Universal Robots PolyScope program: grpB222.urp

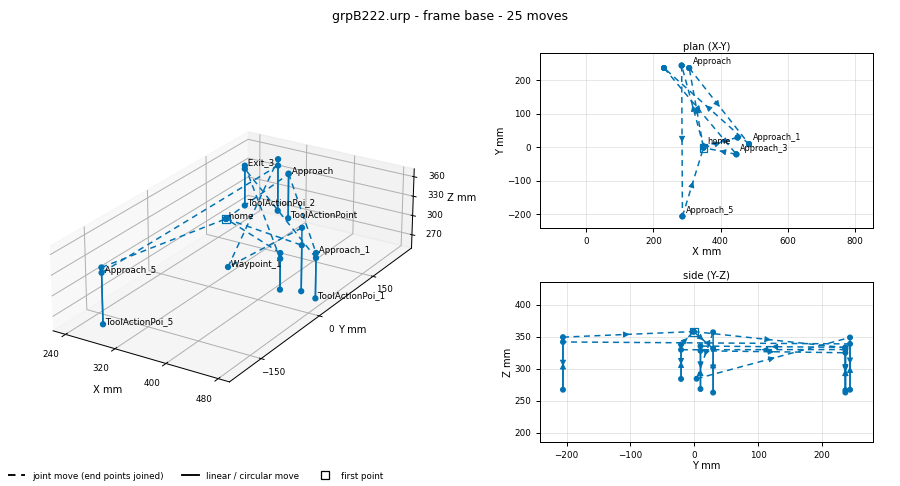
[picture p0: tool path of grpB222.urp in frame base, 25 of 25 moves have a stored position in this frame; points joined in program order, loops and branches not executed]
Program grpB222 (installation=default directory=/programs/Students createdIn=5.11.9.1010452 lastSavedIn=5.11.9.1010452 robotSerialNumber=20225200364)
Calibrated DH parameters: a=[0.00002, -0.569483, -0.54992, -0.00001, -0.000036, 0]; d=[0.180894, -146.691669, 192.918669, -46.053088, 0.119778, 0.115602]; alpha=[1.571425, -0.001534, 0.003359, 1.568739, -1.571477, 0]; deltaTheta=[0, 0.376258, -0.101074, -0.275185, -0.000002, 0]
Robot Program (runOnlyOnce=false)
  MoveJ speed 60 deg/s, acceleration 80 deg/s^2 (useActiveTCP=true) feature=Base
    Waypoint home: TCP in base x=349.211 y=-1.072 z=358.337 mm, rx=2.2343 ry=-2.1885 rz=-0.0245 rad; joints [29.524, -85.445, -128.627, -236.977, -90.829, -151.415] deg
    URCap RG Grip (OnRobot, OnRobot A/S) dataModel(rg-target-force=40.0, rg-target-width=0.1014, Variable(key=on_return, variable(name=on_return)))
    Loop Counting (count=3) loopVariable(name=Loop_1)
      URCap Palletizing (polyscope-pallet-impl, Universal Robots) dataModel(palletFeature=Base, isPalletizing=true, Variable(key=name, variable(name=Pallet_1)), Variable(key=globalCountingVariable, variable(name=Pallet_1_cnt_1, initializeExpression=1)), Variable(key=layerNumberVariable, variable(name=Pallet_1_lno, initializeExpression=1)), Variable(key=layerCountingVariable, variable(name=Pallet_1_lct, initializeExpression=1)), Variable(key=handleSeparatorVariable, variable(name=Pallet_1_sep, initializeExpression=False)), Variable(key=totalCountVariable, variable(name=Pallet_1_tct, initializeExpression=1)), Length(key=objectHeight value=0.00001 unit=M), Variable(key=referencePoint, variable(featureName=referencePoint)), Variable(key=separatorPoint, variable(featureName=separatorPoint))); state(isChildrenLocked=true)
        URCap Patterns (polyscope-pallet-impl, Universal Robots) state(isChildrenLocked=true)
          URCap Pattern (polyscope-pallet-impl, Universal Robots) dataModel(UUID=d454d891-f643-4f11-adf8-96f27634d373, patternType=LINE, objects=3, Variable(key=nameVariable, variable(name=Line_Pattern_1))); state(isChildrenLocked=true)
            URCap Item (polyscope-pallet-impl, Universal Robots) dataModel(UUID=64ea6bed-dd7c-44ae-b121-99742a1ae98b, patternType=LINE, index=0, calibrationDeltaTheta=[-2.1094217540068572E-7, 0.37625772532806073, -0.10107441100396769, -0.2751850025766889, -1.8024952768980196E-6, 2.9402326063437956E-8], calibrationA=[2.0416891277915125E-5, -0.5694828868469309, -0.5499202125525207, -9.504674691390763E-6, -3.603723657207661E-5, 0.0], calibrationD=[0.1808937726775539, -146.69166934821124, 192.91866861971778, -46.05308757405963, 0.11977780403821288, 0.11560212559305974], calibrationAlpha=[1.5714252480212174, -0.0015337665762078037, 0.0033588312559612306, 1.5687392298942362, -1.5714772428732047, 0.0], calibrationJointChecksum=[-1490546360, -1456574554, -1506622700, -1493399207, -1492840923, -1492940558], calibrationStatus=2, calibrationValidChecksum=true, baseToFeature=[0.0, 0.0, 0.0, 0.0, 0.0, 0.0], TCPOffset=[-6.479107609730361E-6, -2.1640648664167372E-6, 6.459965172400661E-6, -7.466567837094426E-7, 6.496160494327226E-6, 1.4031189272003694E-5], Variable(key=variable, variable(name=StartItem_1)), JointPositions(key=jointpositions, JointPosition(key=[1], Angle(key=pos value=1.117784 unit=RAD)), JointPosition(key=[2], Angle(key=pos value=-1.682038 unit=RAD)), JointPosition(key=[3], Angle(key=pos value=-2.256967 unit=RAD)), JointPosition(key=[4], Angle(key=pos value=-3.923758 unit=RAD)), JointPosition(key=[5], Angle(key=pos value=-1.592734 unit=RAD)), JointPosition(key=[6], Angle(key=pos value=-2.039439 unit=RAD))))
            URCap Item (polyscope-pallet-impl, Universal Robots) dataModel(UUID=acc9778f-9bc3-49a4-a915-6e2dc52f2b95, patternType=LINE, index=1, calibrationDeltaTheta=[-2.1094217540068572E-7, 0.37625772532806073, -0.10107441100396769, -0.2751850025766889, -1.8024952768980196E-6, 2.9402326063437956E-8], calibrationA=[2.0416891277915125E-5, -0.5694828868469309, -0.5499202125525207, -9.504674691390763E-6, -3.603723657207661E-5, 0.0], calibrationD=[0.1808937726775539, -146.69166934821124, 192.91866861971778, -46.05308757405963, 0.11977780403821288, 0.11560212559305974], calibrationAlpha=[1.5714252480212174, -0.0015337665762078037, 0.0033588312559612306, 1.5687392298942362, -1.5714772428732047, 0.0], calibrationJointChecksum=[-1490546360, -1456574554, -1506622700, -1493399207, -1492840923, -1492940558], calibrationStatus=2, calibrationValidChecksum=true, baseToFeature=[0.0, 0.0, 0.0, 0.0, 0.0, 0.0], TCPOffset=[1.9374486620010734E-5, 1.7322688802723363E-5, 1.403770617985911E-5, -2.993389842851144E-5, 5.83636955800167E-5, -2.7174622035027854E-5], Variable(key=variable, variable(name=EndItem_1)), JointPositions(key=jointpositions, JointPosition(key=[1], Angle(key=pos value=1.274188 unit=RAD)), JointPosition(key=[2], Angle(key=pos value=-1.609872 unit=RAD)), JointPosition(key=[3], Angle(key=pos value=-2.336948 unit=RAD)), JointPosition(key=[4], Angle(key=pos value=-3.912921 unit=RAD)), JointPosition(key=[5], Angle(key=pos value=-1.593886 unit=RAD)), JointPosition(key=[6], Angle(key=pos value=-1.883026 unit=RAD))))
        URCap Layers (polyscope-pallet-impl, Universal Robots) dataModel(separators=[false], selectedPatterns=[d454d891-f643-4f11-adf8-96f27634d373])
        URCap At Each Item (polyscope-pallet-impl, Universal Robots) dataModel(selectedPattern=d454d891-f643-4f11-adf8-96f27634d373, selectedPosition=64ea6bed-dd7c-44ae-b121-99742a1ae98b, Approach_calibrationDeltaTheta=[-2.1094217540068572E-7, 0.37625772532806073, -0.10107441100396769, -0.2751850025766889, -1.8024952768980196E-6, 2.9402326063437956E-8], Approach_calibrationA=[2.0416891277915125E-5, -0.5694828868469309, -0.5499202125525207, -9.504674691390763E-6, -3.603723657207661E-5, 0.0], Approach_calibrationD=[0.1808937726775539, -146.69166934821124, 192.91866861971778, -46.05308757405963, 0.11977780403821288, 0.11560212559305974], Approach_calibrationAlpha=[1.5714252480212174, -0.0015337665762078037, 0.0033588312559612306, 1.5687392298942362, -1.5714772428732047, 0.0], Approach_calibrationJointChecksum=[-1490546360, -1456574554, -1506622700, -1493399207, -1492840923, -1492940558], Approach_calibrationStatus=2, Approach_calibrationValidChecksum=true, Approach_baseToFeature=[0.0, 0.0, 0.0, 0.0, 0.0, 0.0], Approach_TCPOffset=[2.5781352005288527E-5, 2.5671739316002196E-6, 1.3650458078329208E-5, -3.390166594725408E-5, 6.308214025204194E-5, 7.147033976335445E-5], Exit_calibrationDeltaTheta=[-2.1094217540068572E-7, 0.37625772532806073, -0.10107441100396769, -0.2751850025766889, -1.8024952768980196E-6, 2.9402326063437956E-8], Exit_calibrationA=[2.0416891277915125E-5, -0.5694828868469309, -0.5499202125525207, -9.504674691390763E-6, -3.603723657207661E-5, 0.0], Exit_calibrationD=[0.1808937726775539, -146.69166934821124, 192.91866861971778, -46.05308757405963, 0.11977780403821288, 0.11560212559305974], Exit_calibrationAlpha=[1.5714252480212174, -0.0015337665762078037, 0.0033588312559612306, 1.5687392298942362, -1.5714772428732047, 0.0], Exit_calibrationJointChecksum=[-1490546360, -1456574554, -1506622700, -1493399207, -1492840923, -1492940558], Exit_calibrationStatus=2, Exit_calibrationValidChecksum=true, Exit_baseToFeature=[0.0, 0.0, 0.0, 0.0, 0.0, 0.0], Exit_TCPOffset=[4.769778841942629E-5, 1.539205112810471E-5, 1.24869559859353E-5, -7.939274321106401E-5, 8.864952215778513E-5, 6.565241233819079E-5], currentWizardState=SHOW_DONE, Pose(key=refBaseToFeature, Position(key=posePosition, Length(key=X value=0 unit=M), Length(key=Y value=0 unit=M), Length(key=Z value=0 unit=M)), Rotation(key=poseRotation, Angle(key=RX value=0 unit=RAD), Angle(key=RY value=0 unit=RAD), Angle(key=RZ value=0 unit=RAD))), Pose(key=refPose, Position(key=posePosition, Length(key=X value=0.306641 unit=M), Length(key=Y value=0.236656 unit=M), Length(key=Z value=0.26283 unit=M)), Rotation(key=poseRotation, Angle(key=RX value=2.234367 unit=RAD), Angle(key=RY value=-2.188526 unit=RAD), Angle(key=RZ value=-0.024467 unit=RAD))), JointPositions(key=Approach_jointpositions, JointPosition(key=[1], Angle(key=pos value=1.117614 unit=RAD)), JointPosition(key=[2], Angle(key=pos value=-1.591367 unit=RAD)), JointPosition(key=[3], Angle(key=pos value=-2.200898 unit=RAD)), JointPosition(key=[4], Angle(key=pos value=-4.07051 unit=RAD)), JointPosition(key=[5], Angle(key=pos value=-1.593074 unit=RAD)), JointPosition(key=[6], Angle(key=pos value=-2.040098 unit=RAD))), JointPositions(key=Exit_jointpositions, JointPosition(key=[1], Angle(key=pos value=1.117612 unit=RAD)), JointPosition(key=[2], Angle(key=pos value=-1.590509 unit=RAD)), JointPosition(key=[3], Angle(key=pos value=-2.200233 unit=RAD)), JointPosition(key=[4], Angle(key=pos value=-4.072033 unit=RAD)), JointPosition(key=[5], Angle(key=pos value=-1.593077 unit=RAD)), JointPosition(key=[6], Angle(key=pos value=-2.040105 unit=RAD))))
          URCap Generated Movements (polyscope-pallet-impl, Universal Robots) state(isChildrenLocked=true)
            MoveJ speed 60 deg/s, acceleration 80 deg/s^2 (useActiveTCP=true) feature=referencePoint
              Waypoint Approach: TCP in base x=306.638 y=236.63 z=332.959 mm, rx=2.2342 ry=-2.1886 rz=-0.0244 rad; joints [64.033, -91.179, -126.104, -233.224, -91.277, -116.887] deg; TCP offset x=0 y=0 z=0 mm, rx=0 ry=0 rz=0 rad; feature pose in base x=306.641 y=236.656 z=262.83 mm, rx=2.2344 ry=-2.1885 rz=-0.0245 rad
            MoveL speed 250 mm/s, acceleration 1200 mm/s^2 (useActiveTCP=true) feature(featureName=referencePoint)
              Waypoint ToolActionPoint: TCP in base x=306.641 y=236.656 z=262.83 mm, rx=2.2344 ry=-2.1885 rz=-0.0245 rad; joints [64.045, -96.692, -129.469, -224.342, -91.256, -116.849] deg; TCP offset x=0 y=0 z=0 mm, rx=0 ry=0 rz=0 rad
            Folder Tool action
              URCap RG Grip (OnRobot, OnRobot A/S) dataModel(rg-target-force=40.0, rg-target-width=0.0747)
            MoveL speed 250 mm/s, acceleration 1200 mm/s^2 (useActiveTCP=true) feature(featureName=referencePoint)
              Waypoint Exit_1: TCP in base x=306.626 y=236.608 z=333.664 mm, rx=2.2342 ry=-2.1885 rz=-0.0245 rad; joints [64.033, -91.128, -126.068, -233.314, -91.278, -116.888] deg; TCP offset x=0 y=0 z=0 mm, rx=0 ry=0 rz=0 rad
      URCap Palletizing (polyscope-pallet-impl, Universal Robots) dataModel(palletFeature=Base, isPalletizing=true, Length(key=objectHeight value=0.00001 unit=M), Variable(key=name, variable(name=Pallet_2)), Variable(key=globalCountingVariable, variable(name=Pallet_2_cnt, initializeExpression=1)), Variable(key=layerNumberVariable, variable(name=Pallet_2_lno, initializeExpression=1)), Variable(key=layerCountingVariable, variable(name=Pallet_2_lct, initializeExpression=1)), Variable(key=handleSeparatorVariable, variable(name=Pallet_2_sep, initializeExpression=False)), Variable(key=totalCountVariable, variable(name=Pallet_2_tct, initializeExpression=1)), Variable(key=referencePoint, variable(featureName=referencePoin_1)), Variable(key=separatorPoint, variable(featureName=separatorPoin_1))); state(isChildrenLocked=true)
        URCap Patterns (polyscope-pallet-impl, Universal Robots) state(isChildrenLocked=true)
          URCap Pattern (polyscope-pallet-impl, Universal Robots) dataModel(UUID=45a8ee5b-4a8a-4b28-a838-296028420bac, patternType=LINE, objects=3, Variable(key=nameVariable, variable(name=Line_Pattern_2))); state(isChildrenLocked=true)
            URCap Item (polyscope-pallet-impl, Universal Robots) dataModel(UUID=b27af457-f974-4cfa-a6aa-9b6048d656b7, patternType=LINE, index=0, calibrationDeltaTheta=[-2.1094217540068572E-7, 0.37625772532806073, -0.10107441100396769, -0.2751850025766889, -1.8024952768980196E-6, 2.9402326063437956E-8], calibrationA=[2.0416891277915125E-5, -0.5694828868469309, -0.5499202125525207, -9.504674691390763E-6, -3.603723657207661E-5, 0.0], calibrationD=[0.1808937726775539, -146.69166934821124, 192.91866861971778, -46.05308757405963, 0.11977780403821288, 0.11560212559305974], calibrationAlpha=[1.5714252480212174, -0.0015337665762078037, 0.0033588312559612306, 1.5687392298942362, -1.5714772428732047, 0.0], calibrationJointChecksum=[-1490546360, -1456574554, -1506622700, -1493399207, -1492840923, -1492940558], calibrationStatus=2, calibrationValidChecksum=true, baseToFeature=[0.0, 0.0, 0.0, 0.0, 0.0, 0.0], TCPOffset=[6.044463015194733E-8, 8.449471585958435E-6, 1.7500404647985413E-5, -5.2372560383104365E-6, 3.613439746095069E-5, 5.677349546775118E-6], Variable(key=variable, variable(name=StartItem_2)), JointPositions(key=jointpositions, JointPosition(key=[1], Angle(key=pos value=0.387931 unit=RAD)), JointPosition(key=[2], Angle(key=pos value=-1.834321 unit=RAD)), JointPosition(key=[3], Angle(key=pos value=-2.075058 unit=RAD)), JointPosition(key=[4], Angle(key=pos value=-3.964125 unit=RAD)), JointPosition(key=[5], Angle(key=pos value=-1.582177 unit=RAD)), JointPosition(key=[6], Angle(key=pos value=-2.769248 unit=RAD))))
            URCap Item (polyscope-pallet-impl, Universal Robots) dataModel(UUID=9365cefe-048c-485e-b644-eb1a72d9b5fb, patternType=LINE, index=1, calibrationDeltaTheta=[-2.1094217540068572E-7, 0.37625772532806073, -0.10107441100396769, -0.2751850025766889, -1.8024952768980196E-6, 2.9402326063437956E-8], calibrationA=[2.0416891277915125E-5, -0.5694828868469309, -0.5499202125525207, -9.504674691390763E-6, -3.603723657207661E-5, 0.0], calibrationD=[0.1808937726775539, -146.69166934821124, 192.91866861971778, -46.05308757405963, 0.11977780403821288, 0.11560212559305974], calibrationAlpha=[1.5714252480212174, -0.0015337665762078037, 0.0033588312559612306, 1.5687392298942362, -1.5714772428732047, 0.0], calibrationJointChecksum=[-1490546360, -1456574554, -1506622700, -1493399207, -1492840923, -1492940558], calibrationStatus=2, calibrationValidChecksum=true, baseToFeature=[0.0, 0.0, 0.0, 0.0, 0.0, 0.0], TCPOffset=[-2.5050077170275797E-5, -1.1405127266772563E-5, 6.504272814233936E-7, 1.2865247891813043E-5, -3.7242278860020355E-5, -5.7602559931804165E-5], JointPositions(key=jointpositions, JointPosition(key=[1], Angle(key=pos value=0.44248 unit=RAD)), JointPosition(key=[2], Angle(key=pos value=-1.741933 unit=RAD)), JointPosition(key=[3], Angle(key=pos value=-2.182688 unit=RAD)), JointPosition(key=[4], Angle(key=pos value=-3.948526 unit=RAD)), JointPosition(key=[5], Angle(key=pos value=-1.583418 unit=RAD)), JointPosition(key=[6], Angle(key=pos value=-2.714732 unit=RAD))), Variable(key=variable, variable(name=EndItem_2)))
        URCap Layers (polyscope-pallet-impl, Universal Robots) dataModel(separators=[false], selectedPatterns=[45a8ee5b-4a8a-4b28-a838-296028420bac])
        URCap At Each Item (polyscope-pallet-impl, Universal Robots) dataModel(selectedPattern=45a8ee5b-4a8a-4b28-a838-296028420bac, selectedPosition=b27af457-f974-4cfa-a6aa-9b6048d656b7, Approach_calibrationDeltaTheta=[-2.1094217540068572E-7, 0.37625772532806073, -0.10107441100396769, -0.2751850025766889, -1.8024952768980196E-6, 2.9402326063437956E-8], Approach_calibrationA=[2.0416891277915125E-5, -0.5694828868469309, -0.5499202125525207, -9.504674691390763E-6, -3.603723657207661E-5, 0.0], Approach_calibrationD=[0.1808937726775539, -146.69166934821124, 192.91866861971778, -46.05308757405963, 0.11977780403821288, 0.11560212559305974], Approach_calibrationAlpha=[1.5714252480212174, -0.0015337665762078037, 0.0033588312559612306, 1.5687392298942362, -1.5714772428732047, 0.0], Approach_calibrationJointChecksum=[-1490546360, -1456574554, -1506622700, -1493399207, -1492840923, -1492940558], Approach_calibrationStatus=2, Approach_calibrationValidChecksum=true, Approach_baseToFeature=[0.0, 0.0, 0.0, 0.0, 0.0, 0.0], Approach_TCPOffset=[2.1697404932576178E-5, 2.6992522534685648E-5, 2.5750409892999482E-5, -7.803021143395113E-5, 1.3046438018846386E-5, 5.729013140880056E-5], Exit_calibrationDeltaTheta=[-2.1094217540068572E-7, 0.37625772532806073, -0.10107441100396769, -0.2751850025766889, -1.8024952768980196E-6, 2.9402326063437956E-8], Exit_calibrationA=[2.0416891277915125E-5, -0.5694828868469309, -0.5499202125525207, -9.504674691390763E-6, -3.603723657207661E-5, 0.0], Exit_calibrationD=[0.1808937726775539, -146.69166934821124, 192.91866861971778, -46.05308757405963, 0.11977780403821288, 0.11560212559305974], Exit_calibrationAlpha=[1.5714252480212174, -0.0015337665762078037, 0.0033588312559612306, 1.5687392298942362, -1.5714772428732047, 0.0], Exit_calibrationJointChecksum=[-1490546360, -1456574554, -1506622700, -1493399207, -1492840923, -1492940558], Exit_calibrationStatus=2, Exit_calibrationValidChecksum=true, Exit_baseToFeature=[0.0, 0.0, 0.0, 0.0, 0.0, 0.0], Exit_TCPOffset=[1.9248975832635864E-5, 2.1285860685449354E-5, 4.198514513409357E-5, -9.050769865031771E-5, 5.440701917327053E-5, 1.0746634104783018E-6], currentWizardState=LANDING, Pose(key=refBaseToFeature, Position(key=posePosition, Length(key=X value=0 unit=M), Length(key=Y value=0 unit=M), Length(key=Z value=0 unit=M)), Rotation(key=poseRotation, Angle(key=RX value=0 unit=RAD), Angle(key=RY value=0 unit=RAD), Angle(key=RZ value=0 unit=RAD))), Pose(key=refPose, Position(key=posePosition, Length(key=X value=0.484958 unit=M), Length(key=Y value=0.009632 unit=M), Length(key=Z value=0.268373 unit=M)), Rotation(key=poseRotation, Angle(key=RX value=2.234217 unit=RAD), Angle(key=RY value=-2.1886 unit=RAD), Angle(key=RZ value=-0.024602 unit=RAD))), JointPositions(key=Approach_jointpositions, JointPosition(key=[1], Angle(key=pos value=0.384856 unit=RAD)), JointPosition(key=[2], Angle(key=pos value=-1.753755 unit=RAD)), JointPosition(key=[3], Angle(key=pos value=-2.013529 unit=RAD)), JointPosition(key=[4], Angle(key=pos value=-4.106379 unit=RAD)), JointPosition(key=[5], Angle(key=pos value=-1.582524 unit=RAD)), JointPosition(key=[6], Angle(key=pos value=-2.772795 unit=RAD))), JointPositions(key=Exit_jointpositions, JointPosition(key=[1], Angle(key=pos value=0.384867 unit=RAD)), JointPosition(key=[2], Angle(key=pos value=-1.761546 unit=RAD)), JointPosition(key=[3], Angle(key=pos value=-2.019642 unit=RAD)), JointPosition(key=[4], Angle(key=pos value=-4.092474 unit=RAD)), JointPosition(key=[5], Angle(key=pos value=-1.582497 unit=RAD)), JointPosition(key=[6], Angle(key=pos value=-2.772737 unit=RAD))))
          URCap Generated Movements (polyscope-pallet-impl, Universal Robots) state(isChildrenLocked=true)
            MoveJ speed 60 deg/s, acceleration 80 deg/s^2 (useActiveTCP=true) feature=referencePoin_1
              Waypoint Approach_1: TCP in base x=484.931 y=9.61 z=335.59 mm, rx=2.2341 ry=-2.1886 rz=-0.0247 rad; joints [22.049, -100.483, -115.371, -235.278, -90.673, -158.868] deg; TCP offset x=0 y=0 z=0 mm, rx=0 ry=0 rz=0 rad; feature pose in base x=484.958 y=9.632 z=268.373 mm, rx=2.2342 ry=-2.1886 rz=-0.0246 rad
            MoveL speed 250 mm/s, acceleration 1200 mm/s^2 (useActiveTCP=true) feature(featureName=referencePoin_1)
              Waypoint ToolActionPoi_1: TCP in base x=484.958 y=9.632 z=268.373 mm, rx=2.2342 ry=-2.1886 rz=-0.0246 rad; joints [22.056, -104.961, -118.259, -227.907, -90.656, -158.84] deg; TCP offset x=0 y=0 z=0 mm, rx=0 ry=0 rz=0 rad
            Folder Tool action
              URCap RG Grip (OnRobot, OnRobot A/S) dataModel(rg-target-force=40.0, rg-target-width=0.1014)
            MoveL speed 250 mm/s, acceleration 1200 mm/s^2 (useActiveTCP=true) feature(featureName=referencePoin_1)
              Waypoint Exit_2: TCP in base x=484.936 y=9.612 z=328.275 mm, rx=2.2341 ry=-2.1885 rz=-0.0246 rad; joints [22.05, -100.931, -115.721, -234.481, -90.669, -158.867] deg; TCP offset x=0 y=0 z=0 mm, rx=0 ry=0 rz=0 rad
    Loop Counting (count=3) loopVariable(name=Loop_2)
      URCap Palletizing (polyscope-pallet-impl, Universal Robots) dataModel(palletFeature=Base, isPalletizing=true, Length(key=objectHeight value=0.00001 unit=M), Variable(key=name, variable(name=Pallet_3)), Variable(key=globalCountingVariable, variable(name=Pallet_3_cnt, initializeExpression=1)), Variable(key=layerNumberVariable, variable(name=Pallet_3_lno, initializeExpression=1)), Variable(key=layerCountingVariable, variable(name=Pallet_3_lct, initializeExpression=1)), Variable(key=handleSeparatorVariable, variable(name=Pallet_3_sep, initializeExpression=False)), Variable(key=totalCountVariable, variable(name=Pallet_3_tct, initializeExpression=1)), Variable(key=referencePoint, variable(featureName=referencePoin_2)), Variable(key=separatorPoint, variable(featureName=separatorPoin_2))); state(isChildrenLocked=true)
        URCap Patterns (polyscope-pallet-impl, Universal Robots) state(isChildrenLocked=true)
          URCap Pattern (polyscope-pallet-impl, Universal Robots) dataModel(UUID=2b4160e0-b2a1-4967-a814-10dbe05e682f, patternType=LINE, objects=3, Variable(key=nameVariable, variable(name=Line_Pattern_3))); state(isChildrenLocked=true)
            URCap Item (polyscope-pallet-impl, Universal Robots) dataModel(UUID=27d7fe94-2af4-48ef-bc96-4bf19b8c453b, patternType=LINE, index=0, calibrationDeltaTheta=[-2.1094217540068572E-7, 0.37625772532806073, -0.10107441100396769, -0.2751850025766889, -1.8024952768980196E-6, 2.9402326063437956E-8], calibrationA=[2.0416891277915125E-5, -0.5694828868469309, -0.5499202125525207, -9.504674691390763E-6, -3.603723657207661E-5, 0.0], calibrationD=[0.1808937726775539, -146.69166934821124, 192.91866861971778, -46.05308757405963, 0.11977780403821288, 0.11560212559305974], calibrationAlpha=[1.5714252480212174, -0.0015337665762078037, 0.0033588312559612306, 1.5687392298942362, -1.5714772428732047, 0.0], calibrationJointChecksum=[-1490546360, -1456574554, -1506622700, -1493399207, -1492840923, -1492940558], calibrationStatus=2, calibrationValidChecksum=true, baseToFeature=[0.0, 0.0, 0.0, 0.0, 0.0, 0.0], TCPOffset=[-1.591908718442947E-5, -1.0217043891230793E-5, -2.3879269327009567E-5, 3.6458983264753285E-5, -3.8288802833761E-5, -2.268284047652254E-6], JointPositions(key=jointpositions, JointPosition(key=[1], Angle(key=pos value=1.343103 unit=RAD)), JointPosition(key=[2], Angle(key=pos value=-1.581886 unit=RAD)), JointPosition(key=[3], Angle(key=pos value=-2.365664 unit=RAD)), JointPosition(key=[4], Angle(key=pos value=-3.910843 unit=RAD)), JointPosition(key=[5], Angle(key=pos value=-1.594245 unit=RAD)), JointPosition(key=[6], Angle(key=pos value=-1.814135 unit=RAD))), Variable(key=variable, variable(name=StartItem_3)))
            URCap Item (polyscope-pallet-impl, Universal Robots) dataModel(UUID=072fc38f-4205-41de-a57f-9e135fb71f30, patternType=LINE, index=1, calibrationDeltaTheta=[-2.1094217540068572E-7, 0.37625772532806073, -0.10107441100396769, -0.2751850025766889, -1.8024952768980196E-6, 2.9402326063437956E-8], calibrationA=[2.0416891277915125E-5, -0.5694828868469309, -0.5499202125525207, -9.504674691390763E-6, -3.603723657207661E-5, 0.0], calibrationD=[0.1808937726775539, -146.69166934821124, 192.91866861971778, -46.05308757405963, 0.11977780403821288, 0.11560212559305974], calibrationAlpha=[1.5714252480212174, -0.0015337665762078037, 0.0033588312559612306, 1.5687392298942362, -1.5714772428732047, 0.0], calibrationJointChecksum=[-1490546360, -1456574554, -1506622700, -1493399207, -1492840923, -1492940558], calibrationStatus=2, calibrationValidChecksum=true, baseToFeature=[0.0, 0.0, 0.0, 0.0, 0.0, 0.0], TCPOffset=[-9.716888572375293E-7, -8.226545365752624E-6, -1.2344780305817427E-5, 2.4931859189616642E-5, -3.857283165511878E-5, 3.9017410809858485E-5], JointPositions(key=jointpositions, JointPosition(key=[1], Angle(key=pos value=1.560741 unit=RAD)), JointPosition(key=[2], Angle(key=pos value=-1.505459 unit=RAD)), JointPosition(key=[3], Angle(key=pos value=-2.437569 unit=RAD)), JointPosition(key=[4], Angle(key=pos value=-3.910819 unit=RAD)), JointPosition(key=[5], Angle(key=pos value=-1.59469 unit=RAD)), JointPosition(key=[6], Angle(key=pos value=-1.596497 unit=RAD))), Variable(key=variable, variable(name=EndItem_3)))
        URCap Layers (polyscope-pallet-impl, Universal Robots) dataModel(separators=[false], selectedPatterns=[2b4160e0-b2a1-4967-a814-10dbe05e682f])
        URCap At Each Item (polyscope-pallet-impl, Universal Robots) dataModel(selectedPattern=2b4160e0-b2a1-4967-a814-10dbe05e682f, selectedPosition=27d7fe94-2af4-48ef-bc96-4bf19b8c453b, Approach_calibrationDeltaTheta=[-2.1094217540068572E-7, 0.37625772532806073, -0.10107441100396769, -0.2751850025766889, -1.8024952768980196E-6, 2.9402326063437956E-8], Approach_calibrationA=[2.0416891277915125E-5, -0.5694828868469309, -0.5499202125525207, -9.504674691390763E-6, -3.603723657207661E-5, 0.0], Approach_calibrationD=[0.1808937726775539, -146.69166934821124, 192.91866861971778, -46.05308757405963, 0.11977780403821288, 0.11560212559305974], Approach_calibrationAlpha=[1.5714252480212174, -0.0015337665762078037, 0.0033588312559612306, 1.5687392298942362, -1.5714772428732047, 0.0], Approach_calibrationJointChecksum=[-1490546360, -1456574554, -1506622700, -1493399207, -1492840923, -1492940558], Approach_calibrationStatus=2, Approach_calibrationValidChecksum=true, Approach_baseToFeature=[0.0, 0.0, 0.0, 0.0, 0.0, 0.0], Approach_TCPOffset=[1.671706325981348E-5, -1.0185335574952603E-8, 2.759055502399299E-7, -3.3728848369743684E-5, 2.777383362256239E-5, 1.8955340289357616E-5], Exit_calibrationDeltaTheta=[-2.1094217540068572E-7, 0.37625772532806073, -0.10107441100396769, -0.2751850025766889, -1.8024952768980196E-6, 2.9402326063437956E-8], Exit_calibrationA=[2.0416891277915125E-5, -0.5694828868469309, -0.5499202125525207, -9.504674691390763E-6, -3.603723657207661E-5, 0.0], Exit_calibrationD=[0.1808937726775539, -146.69166934821124, 192.91866861971778, -46.05308757405963, 0.11977780403821288, 0.11560212559305974], Exit_calibrationAlpha=[1.5714252480212174, -0.0015337665762078037, 0.0033588312559612306, 1.5687392298942362, -1.5714772428732047, 0.0], Exit_calibrationJointChecksum=[-1490546360, -1456574554, -1506622700, -1493399207, -1492840923, -1492940558], Exit_calibrationStatus=2, Exit_calibrationValidChecksum=true, Exit_baseToFeature=[0.0, 0.0, 0.0, 0.0, 0.0, 0.0], Exit_TCPOffset=[-1.8147999462536646E-5, -1.7834438799657626E-6, -3.119001539431121E-6, 6.523532778523946E-6, -4.4164474940506126E-5, 2.1790194635512727E-5], currentWizardState=LANDING, Pose(key=refBaseToFeature, Position(key=posePosition, Length(key=X value=0 unit=M), Length(key=Y value=0 unit=M), Length(key=Z value=0 unit=M)), Rotation(key=poseRotation, Angle(key=RX value=0 unit=RAD), Angle(key=RY value=0 unit=RAD), Angle(key=RZ value=0 unit=RAD))), Pose(key=refPose, Position(key=posePosition, Length(key=X value=0.231461 unit=M), Length(key=Y value=0.236677 unit=M), Length(key=Z value=0.266372 unit=M)), Rotation(key=poseRotation, Angle(key=RX value=2.234349 unit=RAD), Angle(key=RY value=-2.188413 unit=RAD), Angle(key=RZ value=-0.024415 unit=RAD))), JointPositions(key=Approach_jointpositions, JointPosition(key=[1], Angle(key=pos value=1.342865 unit=RAD)), JointPosition(key=[2], Angle(key=pos value=-1.492748 unit=RAD)), JointPosition(key=[3], Angle(key=pos value=-2.31193 unit=RAD)), JointPosition(key=[4], Angle(key=pos value=-4.053683 unit=RAD)), JointPosition(key=[5], Angle(key=pos value=-1.594554 unit=RAD)), JointPosition(key=[6], Angle(key=pos value=-1.81486 unit=RAD))), JointPositions(key=Exit_jointpositions, JointPosition(key=[1], Angle(key=pos value=1.342844 unit=RAD)), JointPosition(key=[2], Angle(key=pos value=-1.485893 unit=RAD)), JointPosition(key=[3], Angle(key=pos value=-2.306768 unit=RAD)), JointPosition(key=[4], Angle(key=pos value=-4.065702 unit=RAD)), JointPosition(key=[5], Angle(key=pos value=-1.594578 unit=RAD)), JointPosition(key=[6], Angle(key=pos value=-1.814923 unit=RAD))))
          URCap Generated Movements (polyscope-pallet-impl, Universal Robots) state(isChildrenLocked=true)
            MoveJ speed 60 deg/s, acceleration 80 deg/s^2 (useActiveTCP=true) feature=referencePoin_2
              Waypoint Approach_2: TCP in base x=231.462 y=236.661 z=325.114 mm, rx=2.2343 ry=-2.1884 rz=-0.0244 rad; joints [76.939, -85.528, -132.465, -232.26, -91.363, -103.984] deg; TCP offset x=0 y=0 z=0 mm, rx=0 ry=0 rz=0 rad; feature pose in base x=231.461 y=236.677 z=266.372 mm, rx=2.2343 ry=-2.1884 rz=-0.0244 rad
            MoveL speed 250 mm/s, acceleration 1200 mm/s^2 (useActiveTCP=true) feature(featureName=referencePoin_2)
              Waypoint ToolActionPoi_2: TCP in base x=231.461 y=236.677 z=266.372 mm, rx=2.2343 ry=-2.1884 rz=-0.0244 rad; joints [76.953, -90.634, -135.54, -224.076, -91.342, -103.943] deg; TCP offset x=0 y=0 z=0 mm, rx=0 ry=0 rz=0 rad
            Folder Tool action
              URCap RG Grip (OnRobot, OnRobot A/S) dataModel(rg-target-force=40.0, rg-target-width=0.07440000000000001)
            MoveL speed 250 mm/s, acceleration 1200 mm/s^2 (useActiveTCP=true) feature(featureName=referencePoin_2)
              Waypoint Exit_3: TCP in base x=231.463 y=236.696 z=330.217 mm, rx=2.2344 ry=-2.1885 rz=-0.0245 rad; joints [76.94, -85.136, -132.167, -232.946, -91.363, -103.986] deg; TCP offset x=0 y=0 z=0 mm, rx=0 ry=0 rz=0 rad
      URCap Palletizing (polyscope-pallet-impl, Universal Robots) dataModel(palletFeature=Base, isPalletizing=true, Length(key=objectHeight value=0.00001 unit=M), Variable(key=name, variable(name=Pallet_4)), Variable(key=globalCountingVariable, variable(name=Pallet_4_cnt, initializeExpression=1)), Variable(key=layerNumberVariable, variable(name=Pallet_4_lno, initializeExpression=1)), Variable(key=layerCountingVariable, variable(name=Pallet_4_lct, initializeExpression=1)), Variable(key=handleSeparatorVariable, variable(name=Pallet_4_sep, initializeExpression=False)), Variable(key=totalCountVariable, variable(name=Pallet_4_tct, initializeExpression=1)), Variable(key=referencePoint, variable(featureName=referencePoin_3)), Variable(key=separatorPoint, variable(featureName=separatorPoin_3))); state(isChildrenLocked=true)
        URCap Patterns (polyscope-pallet-impl, Universal Robots) state(isChildrenLocked=true)
          URCap Pattern (polyscope-pallet-impl, Universal Robots) dataModel(UUID=b2d197e2-4b1a-4a96-a263-4bbd625d5d89, patternType=LINE, objects=3, Variable(key=nameVariable, variable(name=Line_Pattern_4))); state(isChildrenLocked=true)
            URCap Item (polyscope-pallet-impl, Universal Robots) dataModel(UUID=846187a8-ace0-42c5-83fe-d86d527c3959, patternType=LINE, index=0, calibrationDeltaTheta=[-2.1094217540068572E-7, 0.37625772532806073, -0.10107441100396769, -0.2751850025766889, -1.8024952768980196E-6, 2.9402326063437956E-8], calibrationA=[2.0416891277915125E-5, -0.5694828868469309, -0.5499202125525207, -9.504674691390763E-6, -3.603723657207661E-5, 0.0], calibrationD=[0.1808937726775539, -146.69166934821124, 192.91866861971778, -46.05308757405963, 0.11977780403821288, 0.11560212559305974], calibrationAlpha=[1.5714252480212174, -0.0015337665762078037, 0.0033588312559612306, 1.5687392298942362, -1.5714772428732047, 0.0], calibrationJointChecksum=[-1490546360, -1456574554, -1506622700, -1493399207, -1492840923, -1492940558], calibrationStatus=2, calibrationValidChecksum=true, baseToFeature=[0.0, 0.0, 0.0, 0.0, 0.0, 0.0], TCPOffset=[6.8659543621119035E-6, -1.6304247807585187E-5, 2.308766209951907E-5, 4.623515782012146E-6, -1.1150474139498562E-5, 1.5743093555091386E-5], Variable(key=variable, variable(name=StartItem_4)), JointPositions(key=jointpositions, JointPosition(key=[1], Angle(key=pos value=0.338559 unit=RAD)), JointPosition(key=[2], Angle(key=pos value=-1.753123 unit=RAD)), JointPosition(key=[3], Angle(key=pos value=-2.133508 unit=RAD)), JointPosition(key=[4], Angle(key=pos value=-3.952628 unit=RAD)), JointPosition(key=[5], Angle(key=pos value=-1.591139 unit=RAD)), JointPosition(key=[6], Angle(key=pos value=-1.227033 unit=RAD))))
            URCap Item (polyscope-pallet-impl, Universal Robots) dataModel(UUID=a6a6b95e-7e2e-4a62-835c-3c2d62c05f01, patternType=LINE, index=1, calibrationDeltaTheta=[-2.1094217540068572E-7, 0.37625772532806073, -0.10107441100396769, -0.2751850025766889, -1.8024952768980196E-6, 2.9402326063437956E-8], calibrationA=[2.0416891277915125E-5, -0.5694828868469309, -0.5499202125525207, -9.504674691390763E-6, -3.603723657207661E-5, 0.0], calibrationD=[0.1808937726775539, -146.69166934821124, 192.91866861971778, -46.05308757405963, 0.11977780403821288, 0.11560212559305974], calibrationAlpha=[1.5714252480212174, -0.0015337665762078037, 0.0033588312559612306, 1.5687392298942362, -1.5714772428732047, 0.0], calibrationJointChecksum=[-1490546360, -1456574554, -1506622700, -1493399207, -1492840923, -1492940558], calibrationStatus=2, calibrationValidChecksum=true, baseToFeature=[0.0, 0.0, 0.0, 0.0, 0.0, 0.0], TCPOffset=[-2.2767164154502417E-6, -8.420508680745398E-6, 5.5903696871695274E-6, -3.318026205864838E-5, 1.717776708781955E-5, 7.755836147888123E-5], Variable(key=variable, variable(name=EndItem_4)), JointPositions(key=jointpositions, JointPosition(key=[1], Angle(key=pos value=0.471697 unit=RAD)), JointPosition(key=[2], Angle(key=pos value=-1.753241 unit=RAD)), JointPosition(key=[3], Angle(key=pos value=-2.132785 unit=RAD)), JointPosition(key=[4], Angle(key=pos value=-3.951055 unit=RAD)), JointPosition(key=[5], Angle(key=pos value=-1.588944 unit=RAD)), JointPosition(key=[6], Angle(key=pos value=-1.093792 unit=RAD))))
        URCap Layers (polyscope-pallet-impl, Universal Robots) dataModel(separators=[false], selectedPatterns=[b2d197e2-4b1a-4a96-a263-4bbd625d5d89])
        URCap At Each Item (polyscope-pallet-impl, Universal Robots) dataModel(selectedPattern=b2d197e2-4b1a-4a96-a263-4bbd625d5d89, selectedPosition=846187a8-ace0-42c5-83fe-d86d527c3959, Approach_calibrationDeltaTheta=[-2.1094217540068572E-7, 0.37625772532806073, -0.10107441100396769, -0.2751850025766889, -1.8024952768980196E-6, 2.9402326063437956E-8], Approach_calibrationA=[2.0416891277915125E-5, -0.5694828868469309, -0.5499202125525207, -9.504674691390763E-6, -3.603723657207661E-5, 0.0], Approach_calibrationD=[0.1808937726775539, -146.69166934821124, 192.91866861971778, -46.05308757405963, 0.11977780403821288, 0.11560212559305974], Approach_calibrationAlpha=[1.5714252480212174, -0.0015337665762078037, 0.0033588312559612306, 1.5687392298942362, -1.5714772428732047, 0.0], Approach_calibrationJointChecksum=[-1490546360, -1456574554, -1506622700, -1493399207, -1492840923, -1492940558], Approach_calibrationStatus=2, Approach_calibrationValidChecksum=true, Approach_baseToFeature=[0.0, 0.0, 0.0, 0.0, 0.0, 0.0], Approach_TCPOffset=[-8.984231985975644E-6, 7.994735703445097E-6, -3.0481751990385497E-5, -5.4916867890803116E-5, -5.758846260962958E-5, 3.04427689044716E-5], Exit_calibrationDeltaTheta=[-2.1094217540068572E-7, 0.37625772532806073, -0.10107441100396769, -0.2751850025766889, -1.8024952768980196E-6, 2.9402326063437956E-8], Exit_calibrationA=[2.0416891277915125E-5, -0.5694828868469309, -0.5499202125525207, -9.504674691390763E-6, -3.603723657207661E-5, 0.0], Exit_calibrationD=[0.1808937726775539, -146.69166934821124, 192.91866861971778, -46.05308757405963, 0.11977780403821288, 0.11560212559305974], Exit_calibrationAlpha=[1.5714252480212174, -0.0015337665762078037, 0.0033588312559612306, 1.5687392298942362, -1.5714772428732047, 0.0], Exit_calibrationJointChecksum=[-1490546360, -1456574554, -1506622700, -1493399207, -1492840923, -1492940558], Exit_calibrationStatus=2, Exit_calibrationValidChecksum=true, Exit_baseToFeature=[0.0, 0.0, 0.0, 0.0, 0.0, 0.0], Exit_TCPOffset=[-7.734931457559213E-6, 8.93221573618555E-6, 4.929908384465609E-6, 2.9480602071985955E-5, -3.2362374490101736E-5, -9.411428258663251E-6], currentWizardState=LANDING, Pose(key=refBaseToFeature, Position(key=posePosition, Length(key=X value=0 unit=M), Length(key=Y value=0 unit=M), Length(key=Z value=0 unit=M)), Rotation(key=poseRotation, Angle(key=RX value=0 unit=RAD), Angle(key=RY value=0 unit=RAD), Angle(key=RZ value=0 unit=RAD))), Pose(key=refPose, Position(key=posePosition, Length(key=X value=0.447307 unit=M), Length(key=Y value=-0.020807 unit=M), Length(key=Z value=0.284151 unit=M)), Rotation(key=poseRotation, Angle(key=RX value=0.000076 unit=RAD), Angle(key=RY value=3.132902 unit=RAD), Angle(key=RZ value=0.034119 unit=RAD))), JointPositions(key=Approach_jointpositions, JointPosition(key=[1], Angle(key=pos value=0.34824 unit=RAD)), JointPosition(key=[2], Angle(key=pos value=-1.690679 unit=RAD)), JointPosition(key=[3], Angle(key=pos value=-2.093004 unit=RAD)), JointPosition(key=[4], Angle(key=pos value=-4.055458 unit=RAD)), JointPosition(key=[5], Angle(key=pos value=-1.591216 unit=RAD)), JointPosition(key=[6], Angle(key=pos value=-1.217596 unit=RAD))), JointPositions(key=Exit_jointpositions, JointPosition(key=[1], Angle(key=pos value=0.348224 unit=RAD)), JointPosition(key=[2], Angle(key=pos value=-1.681442 unit=RAD)), JointPosition(key=[3], Angle(key=pos value=-2.0856 unit=RAD)), JointPosition(key=[4], Angle(key=pos value=-4.0721 unit=RAD)), JointPosition(key=[5], Angle(key=pos value=-1.59125 unit=RAD)), JointPosition(key=[6], Angle(key=pos value=-1.217667 unit=RAD))))
          URCap Generated Movements (polyscope-pallet-impl, Universal Robots) state(isChildrenLocked=true)
            MoveJ speed 60 deg/s, acceleration 80 deg/s^2 (useActiveTCP=true) feature=referencePoin_3
              Waypoint Approach_3: TCP in base x=447.315 y=-20.799 z=329.805 mm, rx=0.0001 ry=3.1328 rz=0.0342 rad; joints [19.953, -96.866, -119.918, -232.361, -91.172, -69.761] deg; TCP offset x=0 y=0 z=0 mm, rx=0 ry=0 rz=0 rad; feature pose in base x=447.307 y=-20.807 z=284.151 mm, rx=0.0001 ry=3.1329 rz=0.0341 rad
            MoveL speed 250 mm/s, acceleration 1200 mm/s^2 (useActiveTCP=true) feature(featureName=referencePoin_3)
              Waypoint ToolActionPoi_3: TCP in base x=447.307 y=-20.807 z=284.151 mm, rx=0.0001 ry=3.1329 rz=0.0341 rad; joints [19.957, -100.024, -122.042, -227.083, -91.158, -69.741] deg; TCP offset x=0 y=0 z=0 mm, rx=0 ry=0 rz=0 rad
            Folder Tool action
              URCap RG Grip (OnRobot, OnRobot A/S) dataModel(rg-target-force=40.0, rg-target-width=0.1014)
            MoveL speed 250 mm/s, acceleration 1200 mm/s^2 (useActiveTCP=true) feature(featureName=referencePoin_3)
              Waypoint Exit_4: TCP in base x=447.314 y=-20.798 z=338.088 mm, rx=0.0001 ry=3.1329 rz=0.0341 rad; joints [19.953, -96.34, -119.496, -233.313, -91.17, -69.766] deg; TCP offset x=0 y=0 z=0 mm, rx=0 ry=0 rz=0 rad
    Waypoint home: TCP in base x=349.211 y=-1.072 z=358.337 mm, rx=2.2343 ry=-2.1885 rz=-0.0245 rad; joints [29.524, -85.445, -128.627, -236.977, -90.829, -151.415] deg
    Loop Counting (count=6) loopVariable(name=Loop_3)
      URCap Palletizing (polyscope-pallet-impl, Universal Robots) dataModel(palletFeature=Base, isPalletizing=false, Length(key=objectHeight value=0.00001 unit=M), Variable(key=name, variable(name=Pallet_6)), Variable(key=globalCountingVariable, variable(name=Pallet_6_cnt, initializeExpression=1)), Variable(key=layerNumberVariable, variable(name=Pallet_6_lno, initializeExpression=1)), Variable(key=layerCountingVariable, variable(name=Pallet_6_lct, initializeExpression=1)), Variable(key=handleSeparatorVariable, variable(name=Pallet_6_sep, initializeExpression=False)), Variable(key=totalCountVariable, variable(name=Pallet_6_tct, initializeExpression=1)), Variable(key=referencePoint, variable(featureName=referencePoin_5)), Variable(key=separatorPoint, variable(featureName=separatorPoin_5))); state(isChildrenLocked=true)
        URCap Patterns (polyscope-pallet-impl, Universal Robots) state(isChildrenLocked=true)
          URCap Pattern (polyscope-pallet-impl, Universal Robots) dataModel(UUID=1c4640bc-86bd-4f4d-a23f-cb4b1a396e7f, patternType=LINE, objects=3, Variable(key=nameVariable, variable(name=Line_Pattern_6))); state(isChildrenLocked=true)
            URCap Item (polyscope-pallet-impl, Universal Robots) dataModel(UUID=00b24ca2-0ee1-4350-97aa-a83631b79931, patternType=LINE, index=0, calibrationDeltaTheta=[-2.1094217540068572E-7, 0.37625772532806073, -0.10107441100396769, -0.2751850025766889, -1.8024952768980196E-6, 2.9402326063437956E-8], calibrationA=[2.0416891277915125E-5, -0.5694828868469309, -0.5499202125525207, -9.504674691390763E-6, -3.603723657207661E-5, 0.0], calibrationD=[0.1808937726775539, -146.69166934821124, 192.91866861971778, -46.05308757405963, 0.11977780403821288, 0.11560212559305974], calibrationAlpha=[1.5714252480212174, -0.0015337665762078037, 0.0033588312559612306, 1.5687392298942362, -1.5714772428732047, 0.0], calibrationJointChecksum=[-1490546360, -1456574554, -1506622700, -1493399207, -1492840923, -1492940558], calibrationStatus=2, calibrationValidChecksum=true, baseToFeature=[0.0, 0.0, 0.0, 0.0, 0.0, 0.0], TCPOffset=[3.666318932571411E-5, -3.103407806931413E-5, 1.4123156632572798E-5, 8.144942798501456E-6, 7.985598922683092E-5, 8.961289321952144E-5], Variable(key=variable, variable(name=StartItem_6)), JointPositions(key=jointpositions, JointPosition(key=[1], Angle(key=pos value=0.451004 unit=RAD)), JointPosition(key=[2], Angle(key=pos value=-1.760458 unit=RAD)), JointPosition(key=[3], Angle(key=pos value=-2.125557 unit=RAD)), JointPosition(key=[4], Angle(key=pos value=-3.948082 unit=RAD)), JointPosition(key=[5], Angle(key=pos value=-1.609128 unit=RAD)), JointPosition(key=[6], Angle(key=pos value=-1.087056 unit=RAD))))
            URCap Item (polyscope-pallet-impl, Universal Robots) dataModel(UUID=03e75c4c-f30b-493e-9341-b5e5fcdd1f91, patternType=LINE, index=1, calibrationDeltaTheta=[-2.1094217540068572E-7, 0.37625772532806073, -0.10107441100396769, -0.2751850025766889, -1.8024952768980196E-6, 2.9402326063437956E-8], calibrationA=[2.0416891277915125E-5, -0.5694828868469309, -0.5499202125525207, -9.504674691390763E-6, -3.603723657207661E-5, 0.0], calibrationD=[0.1808937726775539, -146.69166934821124, 192.91866861971778, -46.05308757405963, 0.11977780403821288, 0.11560212559305974], calibrationAlpha=[1.5714252480212174, -0.0015337665762078037, 0.0033588312559612306, 1.5687392298942362, -1.5714772428732047, 0.0], calibrationJointChecksum=[-1490546360, -1456574554, -1506622700, -1493399207, -1492840923, -1492940558], calibrationStatus=2, calibrationValidChecksum=true, baseToFeature=[0.0, 0.0, 0.0, 0.0, 0.0, 0.0], TCPOffset=[-1.5634672600794985E-5, 1.080114850665441E-5, -3.1264241126538472E-6, -2.7488373969531044E-7, 1.2667663724561166E-5, 2.3999846943894514E-6], Variable(key=variable, variable(name=EndItem_6)), JointPositions(key=jointpositions, JointPosition(key=[1], Angle(key=pos value=0.335745 unit=RAD)), JointPosition(key=[2], Angle(key=pos value=-1.759567 unit=RAD)), JointPosition(key=[3], Angle(key=pos value=-2.12466 unit=RAD)), JointPosition(key=[4], Angle(key=pos value=-3.954104 unit=RAD)), JointPosition(key=[5], Angle(key=pos value=-1.611254 unit=RAD)), JointPosition(key=[6], Angle(key=pos value=-1.202328 unit=RAD))))
          URCap Pattern (polyscope-pallet-impl, Universal Robots) dataModel(UUID=eab0a5fa-a9a5-4de0-adc7-d56ff99146b4, patternType=LINE, objects=3, Variable(key=nameVariable, variable(name=Line_Pattern_7))); state(isChildrenLocked=true)
            URCap Item (polyscope-pallet-impl, Universal Robots) dataModel(UUID=5b0d4488-2f4e-4d66-8128-c261d9e8e3e9, patternType=LINE, index=0, calibrationDeltaTheta=[-2.1094217540068572E-7, 0.37625772532806073, -0.10107441100396769, -0.2751850025766889, -1.8024952768980196E-6, 2.9402326063437956E-8], calibrationA=[2.0416891277915125E-5, -0.5694828868469309, -0.5499202125525207, -9.504674691390763E-6, -3.603723657207661E-5, 0.0], calibrationD=[0.1808937726775539, -146.69166934821124, 192.91866861971778, -46.05308757405963, 0.11977780403821288, 0.11560212559305974], calibrationAlpha=[1.5714252480212174, -0.0015337665762078037, 0.0033588312559612306, 1.5687392298942362, -1.5714772428732047, 0.0], calibrationJointChecksum=[-1490546360, -1456574554, -1506622700, -1493399207, -1492840923, -1492940558], calibrationStatus=2, calibrationValidChecksum=true, baseToFeature=[0.0, 0.0, 0.0, 0.0, 0.0, 0.0], TCPOffset=[-3.1551024677559797E-6, -1.4173821301921574E-5, 1.874568991686032E-5, 4.82821619659131E-5, -1.6804247167123245E-5, 6.31448121466832E-7], Variable(key=variable, variable(name=StartItem_7)), JointPositions(key=jointpositions, JointPosition(key=[1], Angle(key=pos value=0.469103 unit=RAD)), JointPosition(key=[2], Angle(key=pos value=-1.711332 unit=RAD)), JointPosition(key=[3], Angle(key=pos value=-2.220286 unit=RAD)), JointPosition(key=[4], Angle(key=pos value=-3.887287 unit=RAD)), JointPosition(key=[5], Angle(key=pos value=-1.553048 unit=RAD)), JointPosition(key=[6], Angle(key=pos value=0.479029 unit=RAD))))
            URCap Item (polyscope-pallet-impl, Universal Robots) dataModel(UUID=ec6de5b8-6bb2-4132-8a11-ad8d3cdfdd0f, patternType=LINE, index=1, calibrationDeltaTheta=[-2.1094217540068572E-7, 0.37625772532806073, -0.10107441100396769, -0.2751850025766889, -1.8024952768980196E-6, 2.9402326063437956E-8], calibrationA=[2.0416891277915125E-5, -0.5694828868469309, -0.5499202125525207, -9.504674691390763E-6, -3.603723657207661E-5, 0.0], calibrationD=[0.1808937726775539, -146.69166934821124, 192.91866861971778, -46.05308757405963, 0.11977780403821288, 0.11560212559305974], calibrationAlpha=[1.5714252480212174, -0.0015337665762078037, 0.0033588312559612306, 1.5687392298942362, -1.5714772428732047, 0.0], calibrationJointChecksum=[-1490546360, -1456574554, -1506622700, -1493399207, -1492840923, -1492940558], calibrationStatus=2, calibrationValidChecksum=true, baseToFeature=[0.0, 0.0, 0.0, 0.0, 0.0, 0.0], TCPOffset=[1.8244568883128698E-6, -3.01631795984747E-7, 3.9595082005350335E-6, -7.412561655762438E-6, -2.3682067464299316E-5, -1.0710739118289924E-5], Variable(key=variable, variable(name=EndItem_7)), JointPositions(key=jointpositions, JointPosition(key=[1], Angle(key=pos value=0.407605 unit=RAD)), JointPosition(key=[2], Angle(key=pos value=-1.799657 unit=RAD)), JointPosition(key=[3], Angle(key=pos value=-2.107185 unit=RAD)), JointPosition(key=[4], Angle(key=pos value=-3.910872 unit=RAD)), JointPosition(key=[5], Angle(key=pos value=-1.555194 unit=RAD)), JointPosition(key=[6], Angle(key=pos value=0.417511 unit=RAD))))
        URCap Layers (polyscope-pallet-impl, Universal Robots) dataModel(separators=[false, false], selectedPatterns=[eab0a5fa-a9a5-4de0-adc7-d56ff99146b4, 1c4640bc-86bd-4f4d-a23f-cb4b1a396e7f])
        URCap At Each Item (polyscope-pallet-impl, Universal Robots) dataModel(selectedPattern=1c4640bc-86bd-4f4d-a23f-cb4b1a396e7f, selectedPosition=00b24ca2-0ee1-4350-97aa-a83631b79931, Approach_calibrationDeltaTheta=[-2.1094217540068572E-7, 0.37625772532806073, -0.10107441100396769, -0.2751850025766889, -1.8024952768980196E-6, 2.9402326063437956E-8], Approach_calibrationA=[2.0416891277915125E-5, -0.5694828868469309, -0.5499202125525207, -9.504674691390763E-6, -3.603723657207661E-5, 0.0], Approach_calibrationD=[0.1808937726775539, -146.69166934821124, 192.91866861971778, -46.05308757405963, 0.11977780403821288, 0.11560212559305974], Approach_calibrationAlpha=[1.5714252480212174, -0.0015337665762078037, 0.0033588312559612306, 1.5687392298942362, -1.5714772428732047, 0.0], Approach_calibrationJointChecksum=[-1490546360, -1456574554, -1506622700, -1493399207, -1492840923, -1492940558], Approach_calibrationStatus=2, Approach_calibrationValidChecksum=true, Approach_baseToFeature=[0.0, 0.0, 0.0, 0.0, 0.0, 0.0], Approach_TCPOffset=[2.1983287934068674E-5, 2.7092795062966246E-7, 3.5565050371388907E-6, 2.428454658877015E-5, 9.095983351029034E-5, -1.1843430025114945E-5], Exit_calibrationDeltaTheta=[-2.1094217540068572E-7, 0.37625772532806073, -0.10107441100396769, -0.2751850025766889, -1.8024952768980196E-6, 2.9402326063437956E-8], Exit_calibrationA=[2.0416891277915125E-5, -0.5694828868469309, -0.5499202125525207, -9.504674691390763E-6, -3.603723657207661E-5, 0.0], Exit_calibrationD=[0.1808937726775539, -146.69166934821124, 192.91866861971778, -46.05308757405963, 0.11977780403821288, 0.11560212559305974], Exit_calibrationAlpha=[1.5714252480212174, -0.0015337665762078037, 0.0033588312559612306, 1.5687392298942362, -1.5714772428732047, 0.0], Exit_calibrationJointChecksum=[-1490546360, -1456574554, -1506622700, -1493399207, -1492840923, -1492940558], Exit_calibrationStatus=2, Exit_calibrationValidChecksum=true, Exit_baseToFeature=[0.0, 0.0, 0.0, 0.0, 0.0, 0.0], Exit_TCPOffset=[6.786595543040175E-6, -7.701714522904968E-6, -2.6220083860772903E-6, 2.414966828600271E-5, 7.100965439547193E-6, 2.105248435710312E-5], currentWizardState=LANDING, Pose(key=refBaseToFeature, Position(key=posePosition, Length(key=X value=0 unit=M), Length(key=Y value=0 unit=M), Length(key=Z value=0 unit=M)), Rotation(key=poseRotation, Angle(key=RX value=0 unit=RAD), Angle(key=RY value=0 unit=RAD), Angle(key=RZ value=0 unit=RAD))), Pose(key=refPose, Position(key=posePosition, Length(key=X value=0.451126 unit=M), Length(key=Y value=0.029446 unit=M), Length(key=Z value=0.262752 unit=M)), Rotation(key=poseRotation, Angle(key=RX value=0.042778 unit=RAD), Angle(key=RY value=3.138452 unit=RAD), Angle(key=RZ value=0.064485 unit=RAD))), JointPositions(key=Approach_jointpositions, JointPosition(key=[1], Angle(key=pos value=0.450913 unit=RAD)), JointPosition(key=[2], Angle(key=pos value=-1.695593 unit=RAD)), JointPosition(key=[3], Angle(key=pos value=-2.082378 unit=RAD)), JointPosition(key=[4], Angle(key=pos value=-4.056142 unit=RAD)), JointPosition(key=[5], Angle(key=pos value=-1.609381 unit=RAD)), JointPosition(key=[6], Angle(key=pos value=-1.087496 unit=RAD))), JointPositions(key=Exit_jointpositions, JointPosition(key=[1], Angle(key=pos value=0.450865 unit=RAD)), JointPosition(key=[2], Angle(key=pos value=-1.668162 unit=RAD)), JointPosition(key=[3], Angle(key=pos value=-2.058756 unit=RAD)), JointPosition(key=[4], Angle(key=pos value=-4.107203 unit=RAD)), JointPosition(key=[5], Angle(key=pos value=-1.609482 unit=RAD)), JointPosition(key=[6], Angle(key=pos value=-1.087715 unit=RAD))))
          URCap Generated Movements (polyscope-pallet-impl, Universal Robots) state(isChildrenLocked=true)
            MoveJ speed 60 deg/s, acceleration 80 deg/s^2 (useActiveTCP=true) feature=referencePoin_5
              Waypoint Approach_4: TCP in base x=451.104 y=29.447 z=331.487 mm, rx=0.0428 ry=3.1385 rz=0.0645 rad; joints [25.837, -97.15, -119.313, -232.403, -92.212, -62.309] deg; TCP offset x=0 y=0 z=0 mm, rx=0 ry=0 rz=0 rad; feature pose in base x=451.126 y=29.446 z=262.752 mm, rx=0.0428 ry=3.1385 rz=0.0645 rad
            MoveL speed 250 mm/s, acceleration 1200 mm/s^2 (useActiveTCP=true) feature(featureName=referencePoin_5)
              Waypoint ToolActionPoi_4: TCP in base x=451.126 y=29.446 z=262.752 mm, rx=0.0428 ry=3.1385 rz=0.0645 rad; joints [25.842, -101.997, -122.382, -224.481, -92.192, -62.277] deg; TCP offset x=0 y=0 z=0 mm, rx=0 ry=0 rz=0 rad
            Folder Tool action
              URCap RG Grip (OnRobot, OnRobot A/S) dataModel(rg-target-force=40.0, rg-target-width=0.0748)
            MoveL speed 250 mm/s, acceleration 1200 mm/s^2 (useActiveTCP=true) feature(featureName=referencePoin_5)
              Waypoint Exit_5: TCP in base x=451.119 y=29.439 z=357.266 mm, rx=0.0428 ry=3.1385 rz=0.0644 rad; joints [25.832, -95.578, -117.959, -235.326, -92.216, -62.321] deg; TCP offset x=0 y=0 z=0 mm, rx=0 ry=0 rz=0 rad
      Waypoint Waypoint_1: TCP in base x=349.207 y=3.599 z=284.439 mm, rx=2.2343 ry=-2.1885 rz=-0.0245 rad; joints [30.298, -91.159, -132.676, -227.207, -90.824, -150.606] deg
      If analog_in[0]>5
        URCap Palletizing (polyscope-pallet-impl, Universal Robots) dataModel(palletFeature=Base, isPalletizing=true, Length(key=objectHeight value=0.00001 unit=M), Variable(key=name, variable(name=Pallet_5)), Variable(key=globalCountingVariable, variable(name=Pallet_5_cnt, initializeExpression=1)), Variable(key=layerNumberVariable, variable(name=Pallet_5_lno, initializeExpression=1)), Variable(key=layerCountingVariable, variable(name=Pallet_5_lct, initializeExpression=1)), Variable(key=handleSeparatorVariable, variable(name=Pallet_5_sep, initializeExpression=False)), Variable(key=totalCountVariable, variable(name=Pallet_5_tct, initializeExpression=1)), Variable(key=referencePoint, variable(featureName=referencePoin_4)), Variable(key=separatorPoint, variable(featureName=separatorPoin_4))); state(isChildrenLocked=true)
          URCap Patterns (polyscope-pallet-impl, Universal Robots) state(isChildrenLocked=true)
            URCap Pattern (polyscope-pallet-impl, Universal Robots) dataModel(UUID=5c0261e5-ffab-4fd7-8cb2-820f88da817b, patternType=LINE, objects=3, Variable(key=nameVariable, variable(name=Line_Pattern_5))); state(isChildrenLocked=true)
              URCap Item (polyscope-pallet-impl, Universal Robots) dataModel(UUID=76805789-12ae-4a56-8aec-022a15e36e52, patternType=LINE, index=0, calibrationDeltaTheta=[-2.1094217540068572E-7, 0.37625772532806073, -0.10107441100396769, -0.2751850025766889, -1.8024952768980196E-6, 2.9402326063437956E-8], calibrationA=[2.0416891277915125E-5, -0.5694828868469309, -0.5499202125525207, -9.504674691390763E-6, -3.603723657207661E-5, 0.0], calibrationD=[0.1808937726775539, -146.69166934821124, 192.91866861971778, -46.05308757405963, 0.11977780403821288, 0.11560212559305974], calibrationAlpha=[1.5714252480212174, -0.0015337665762078037, 0.0033588312559612306, 1.5687392298942362, -1.5714772428732047, 0.0], calibrationJointChecksum=[-1490546360, -1456574554, -1506622700, -1493399207, -1492840923, -1492940558], calibrationStatus=2, calibrationValidChecksum=true, baseToFeature=[0.0, 0.0, 0.0, 0.0, 0.0, 0.0], TCPOffset=[-4.337050140718057E-6, 9.464252731516964E-7, 1.2058841331430425E-5, 1.5977424164385615E-5, 6.839575977425617E-6, -1.5765846175024105E-6], JointPositions(key=jointpositions, JointPosition(key=[1], Angle(key=pos value=1.207414 unit=RAD)), JointPosition(key=[2], Angle(key=pos value=-1.658917 unit=RAD)), JointPosition(key=[3], Angle(key=pos value=-2.285988 unit=RAD)), JointPosition(key=[4], Angle(key=pos value=-3.931135 unit=RAD)), JointPosition(key=[5], Angle(key=pos value=-1.534071 unit=RAD)), JointPosition(key=[6], Angle(key=pos value=-1.891191 unit=RAD))), Variable(key=variable, variable(name=StartItem_5)))
              URCap Item (polyscope-pallet-impl, Universal Robots) dataModel(UUID=6cedd976-d7c8-47ba-b013-1773a5d1cc4a, patternType=LINE, index=1, calibrationDeltaTheta=[-2.1094217540068572E-7, 0.37625772532806073, -0.10107441100396769, -0.2751850025766889, -1.8024952768980196E-6, 2.9402326063437956E-8], calibrationA=[2.0416891277915125E-5, -0.5694828868469309, -0.5499202125525207, -9.504674691390763E-6, -3.603723657207661E-5, 0.0], calibrationD=[0.1808937726775539, -146.69166934821124, 192.91866861971778, -46.05308757405963, 0.11977780403821288, 0.11560212559305974], calibrationAlpha=[1.5714252480212174, -0.0015337665762078037, 0.0033588312559612306, 1.5687392298942362, -1.5714772428732047, 0.0], calibrationJointChecksum=[-1490546360, -1456574554, -1506622700, -1493399207, -1492840923, -1492940558], calibrationStatus=2, calibrationValidChecksum=true, baseToFeature=[0.0, 0.0, 0.0, 0.0, 0.0, 0.0], TCPOffset=[1.5859399769141413E-5, -5.747238972453328E-6, 5.137893616669054E-6, -8.91584319392297E-6, -1.8819193936408115E-5, -3.6777371429346007E-6], JointPositions(key=jointpositions, JointPosition(key=[1], Angle(key=pos value=1.376034 unit=RAD)), JointPosition(key=[2], Angle(key=pos value=-1.59209 unit=RAD)), JointPosition(key=[3], Angle(key=pos value=-2.361549 unit=RAD)), JointPosition(key=[4], Angle(key=pos value=-3.928708 unit=RAD)), JointPosition(key=[5], Angle(key=pos value=-1.538288 unit=RAD)), JointPosition(key=[6], Angle(key=pos value=-1.722534 unit=RAD))), Variable(key=variable, variable(name=EndItem_5)))
          URCap Layers (polyscope-pallet-impl, Universal Robots) dataModel(separators=[false], selectedPatterns=[5c0261e5-ffab-4fd7-8cb2-820f88da817b])
          URCap At Each Item (polyscope-pallet-impl, Universal Robots) dataModel(selectedPattern=5c0261e5-ffab-4fd7-8cb2-820f88da817b, selectedPosition=76805789-12ae-4a56-8aec-022a15e36e52, Approach_calibrationDeltaTheta=[-2.1094217540068572E-7, 0.37625772532806073, -0.10107441100396769, -0.2751850025766889, -1.8024952768980196E-6, 2.9402326063437956E-8], Approach_calibrationA=[2.0416891277915125E-5, -0.5694828868469309, -0.5499202125525207, -9.504674691390763E-6, -3.603723657207661E-5, 0.0], Approach_calibrationD=[0.1808937726775539, -146.69166934821124, 192.91866861971778, -46.05308757405963, 0.11977780403821288, 0.11560212559305974], Approach_calibrationAlpha=[1.5714252480212174, -0.0015337665762078037, 0.0033588312559612306, 1.5687392298942362, -1.5714772428732047, 0.0], Approach_calibrationJointChecksum=[-1490546360, -1456574554, -1506622700, -1493399207, -1492840923, -1492940558], Approach_calibrationStatus=2, Approach_calibrationValidChecksum=true, Approach_baseToFeature=[0.0, 0.0, 0.0, 0.0, 0.0, 0.0], Approach_TCPOffset=[1.2163195871967014E-5, 4.992991399332958E-6, 2.152133657173927E-5, -2.5782126522660622E-5, 1.983399365329415E-5, 1.610377204797929E-5], Exit_calibrationDeltaTheta=[-2.1094217540068572E-7, 0.37625772532806073, -0.10107441100396769, -0.2751850025766889, -1.8024952768980196E-6, 2.9402326063437956E-8], Exit_calibrationA=[2.0416891277915125E-5, -0.5694828868469309, -0.5499202125525207, -9.504674691390763E-6, -3.603723657207661E-5, 0.0], Exit_calibrationD=[0.1808937726775539, -146.69166934821124, 192.91866861971778, -46.05308757405963, 0.11977780403821288, 0.11560212559305974], Exit_calibrationAlpha=[1.5714252480212174, -0.0015337665762078037, 0.0033588312559612306, 1.5687392298942362, -1.5714772428732047, 0.0], Exit_calibrationJointChecksum=[-1490546360, -1456574554, -1506622700, -1493399207, -1492840923, -1492940558], Exit_calibrationStatus=2, Exit_calibrationValidChecksum=true, Exit_baseToFeature=[0.0, 0.0, 0.0, 0.0, 0.0, 0.0], Exit_TCPOffset=[-9.380114039087006E-6, 2.0136365106004916E-5, 1.3678182375131964E-5, -5.499147997712749E-5, 7.000127186227599E-5, -9.736936579608192E-5], currentWizardState=LANDING, Pose(key=refBaseToFeature, Position(key=posePosition, Length(key=X value=0 unit=M), Length(key=Y value=0 unit=M), Length(key=Z value=0 unit=M)), Rotation(key=poseRotation, Angle(key=RX value=0 unit=RAD), Angle(key=RY value=0 unit=RAD), Angle(key=RZ value=0 unit=RAD))), Pose(key=refPose, Position(key=posePosition, Length(key=X value=0.284198 unit=M), Length(key=Y value=0.243934 unit=M), Length(key=Z value=0.267233 unit=M)), Rotation(key=poseRotation, Angle(key=RX value=2.177405 unit=RAD), Angle(key=RY value=-2.260349 unit=RAD), Angle(key=RZ value=0.070272 unit=RAD))), JointPositions(key=Approach_jointpositions, JointPosition(key=[1], Angle(key=pos value=1.207188 unit=RAD)), JointPosition(key=[2], Angle(key=pos value=-1.547046 unit=RAD)), JointPosition(key=[3], Angle(key=pos value=-2.213746 unit=RAD)), JointPosition(key=[4], Angle(key=pos value=-4.115215 unit=RAD)), JointPosition(key=[5], Angle(key=pos value=-1.534458 unit=RAD)), JointPosition(key=[6], Angle(key=pos value=-1.892046 unit=RAD))), JointPositions(key=Exit_jointpositions, JointPosition(key=[1], Angle(key=pos value=1.20722 unit=RAD)), JointPosition(key=[2], Angle(key=pos value=-1.559176 unit=RAD)), JointPosition(key=[3], Angle(key=pos value=-2.223723 unit=RAD)), JointPosition(key=[4], Angle(key=pos value=-4.093113 unit=RAD)), JointPosition(key=[5], Angle(key=pos value=-1.534417 unit=RAD)), JointPosition(key=[6], Angle(key=pos value=-1.891937 unit=RAD))))
            URCap Generated Movements (polyscope-pallet-impl, Universal Robots) state(isChildrenLocked=true)
              MoveJ speed 60 deg/s, acceleration 80 deg/s^2 (useActiveTCP=true) feature=referencePoin_4
                Waypoint Approach_6: TCP in base x=284.193 y=243.921 z=349.082 mm, rx=2.1774 ry=-2.2603 rz=0.0703 rad; joints [69.166, -88.64, -126.841, -235.783, -87.919, -108.406] deg; TCP offset x=0 y=0 z=0 mm, rx=0 ry=0 rz=0 rad; feature pose in base x=284.198 y=243.934 z=267.233 mm, rx=2.1774 ry=-2.2603 rz=0.0703 rad
              MoveL speed 250 mm/s, acceleration 1200 mm/s^2 (useActiveTCP=true) feature(featureName=referencePoin_4)
                Waypoint ToolActionPoi_6: TCP in base x=284.198 y=243.934 z=267.233 mm, rx=2.1774 ry=-2.2603 rz=0.0703 rad; joints [69.18, -95.05, -130.978, -225.236, -87.895, -108.357] deg; TCP offset x=0 y=0 z=0 mm, rx=0 ry=0 rz=0 rad
              Folder Tool action
                URCap RG Grip (OnRobot, OnRobot A/S) dataModel(rg-target-force=40.0, rg-target-width=0.1014)
              MoveL speed 250 mm/s, acceleration 1200 mm/s^2 (useActiveTCP=true) feature(featureName=referencePoin_4)
                Waypoint Exit_7: TCP in base x=284.178 y=243.944 z=339.008 mm, rx=2.1774 ry=-2.2602 rz=0.0703 rad; joints [69.172, -89.336, -127.411, -234.52, -87.917, -108.402] deg; TCP offset x=0 y=0 z=0 mm, rx=0 ry=0 rz=0 rad
      Else 
        URCap Palletizing (polyscope-pallet-impl, Universal Robots) dataModel(palletFeature=Base, isPalletizing=true, Length(key=objectHeight value=0.00001 unit=M), Variable(key=name, variable(name=Pallet_7)), Variable(key=globalCountingVariable, variable(name=Pallet_7_cnt, initializeExpression=1)), Variable(key=layerNumberVariable, variable(name=Pallet_7_lno, initializeExpression=1)), Variable(key=layerCountingVariable, variable(name=Pallet_7_lct, initializeExpression=1)), Variable(key=handleSeparatorVariable, variable(name=Pallet_7_sep, initializeExpression=False)), Variable(key=totalCountVariable, variable(name=Pallet_7_tct, initializeExpression=1)), Variable(key=referencePoint, variable(featureName=referencePoin_6)), Variable(key=separatorPoint, variable(featureName=separatorPoin_6))); state(isChildrenLocked=true)
          URCap Patterns (polyscope-pallet-impl, Universal Robots) state(isChildrenLocked=true)
            URCap Pattern (polyscope-pallet-impl, Universal Robots) dataModel(UUID=7aca8206-a6f6-4ad4-ae03-99b5f4470156, patternType=LINE, objects=3, Variable(key=nameVariable, variable(name=Line_Pattern_8))); state(isChildrenLocked=true)
              URCap Item (polyscope-pallet-impl, Universal Robots) dataModel(UUID=57d4a94b-b0dd-408c-9eaf-3dcc8e425f30, patternType=LINE, index=0, calibrationDeltaTheta=[-2.1094217540068572E-7, 0.37625772532806073, -0.10107441100396769, -0.2751850025766889, -1.8024952768980196E-6, 2.9402326063437956E-8], calibrationA=[2.0416891277915125E-5, -0.5694828868469309, -0.5499202125525207, -9.504674691390763E-6, -3.603723657207661E-5, 0.0], calibrationD=[0.1808937726775539, -146.69166934821124, 192.91866861971778, -46.05308757405963, 0.11977780403821288, 0.11560212559305974], calibrationAlpha=[1.5714252480212174, -0.0015337665762078037, 0.0033588312559612306, 1.5687392298942362, -1.5714772428732047, 0.0], calibrationJointChecksum=[-1490546360, -1456574554, -1506622700, -1493399207, -1492840923, -1492940558], calibrationStatus=2, calibrationValidChecksum=true, baseToFeature=[0.0, 0.0, 0.0, 0.0, 0.0, 0.0], TCPOffset=[5.793444083607158E-6, -2.921163469038479E-5, -8.859777279157655E-6, 3.915245999676412E-5, 2.7777688418041124E-5, -2.310336838907693E-6], JointPositions(key=jointpositions, JointPosition(key=[1], Angle(key=pos value=-0.093977 unit=RAD)), JointPosition(key=[2], Angle(key=pos value=-1.601309 unit=RAD)), JointPosition(key=[3], Angle(key=pos value=-2.332846 unit=RAD)), JointPosition(key=[4], Angle(key=pos value=-3.888212 unit=RAD)), JointPosition(key=[5], Angle(key=pos value=-1.542586 unit=RAD)), JointPosition(key=[6], Angle(key=pos value=-3.193421 unit=RAD))), Variable(key=variable, variable(name=StartItem_8)))
              URCap Item (polyscope-pallet-impl, Universal Robots) dataModel(UUID=b348cbc8-de4f-4515-9b8b-d1701aeaa393, patternType=LINE, index=1, calibrationDeltaTheta=[-2.1094217540068572E-7, 0.37625772532806073, -0.10107441100396769, -0.2751850025766889, -1.8024952768980196E-6, 2.9402326063437956E-8], calibrationA=[2.0416891277915125E-5, -0.5694828868469309, -0.5499202125525207, -9.504674691390763E-6, -3.603723657207661E-5, 0.0], calibrationD=[0.1808937726775539, -146.69166934821124, 192.91866861971778, -46.05308757405963, 0.11977780403821288, 0.11560212559305974], calibrationAlpha=[1.5714252480212174, -0.0015337665762078037, 0.0033588312559612306, 1.5687392298942362, -1.5714772428732047, 0.0], calibrationJointChecksum=[-1490546360, -1456574554, -1506622700, -1493399207, -1492840923, -1492940558], calibrationStatus=2, calibrationValidChecksum=true, baseToFeature=[0.0, 0.0, 0.0, 0.0, 0.0, 0.0], TCPOffset=[-1.7761107696245837E-6, 7.0185800350452965E-6, -2.9198431213961484E-6, 3.7597373406695815E-5, 1.117454483118892E-5, -1.4785706678834087E-5], Variable(key=variable, variable(name=EndItem_8)), JointPositions(key=jointpositions, JointPosition(key=[1], Angle(key=pos value=-0.114353 unit=RAD)), JointPosition(key=[2], Angle(key=pos value=-1.521226 unit=RAD)), JointPosition(key=[3], Angle(key=pos value=-2.416888 unit=RAD)), JointPosition(key=[4], Angle(key=pos value=-3.883617 unit=RAD)), JointPosition(key=[5], Angle(key=pos value=-1.543381 unit=RAD)), JointPosition(key=[6], Angle(key=pos value=-3.213775 unit=RAD))))
          URCap Layers (polyscope-pallet-impl, Universal Robots) dataModel(separators=[false], selectedPatterns=[7aca8206-a6f6-4ad4-ae03-99b5f4470156])
          URCap At Each Item (polyscope-pallet-impl, Universal Robots) dataModel(selectedPattern=7aca8206-a6f6-4ad4-ae03-99b5f4470156, selectedPosition=57d4a94b-b0dd-408c-9eaf-3dcc8e425f30, Approach_calibrationDeltaTheta=[-2.1094217540068572E-7, 0.37625772532806073, -0.10107441100396769, -0.2751850025766889, -1.8024952768980196E-6, 2.9402326063437956E-8], Approach_calibrationA=[2.0416891277915125E-5, -0.5694828868469309, -0.5499202125525207, -9.504674691390763E-6, -3.603723657207661E-5, 0.0], Approach_calibrationD=[0.1808937726775539, -146.69166934821124, 192.91866861971778, -46.05308757405963, 0.11977780403821288, 0.11560212559305974], Approach_calibrationAlpha=[1.5714252480212174, -0.0015337665762078037, 0.0033588312559612306, 1.5687392298942362, -1.5714772428732047, 0.0], Approach_calibrationJointChecksum=[-1490546360, -1456574554, -1506622700, -1493399207, -1492840923, -1492940558], Approach_calibrationStatus=2, Approach_calibrationValidChecksum=true, Approach_baseToFeature=[0.0, 0.0, 0.0, 0.0, 0.0, 0.0], Approach_TCPOffset=[-6.393256510528467E-6, -1.2309234991680906E-5, 8.454835641213965E-6, -7.3402317364412775E-6, -7.125703807256485E-5, -3.541805901267217E-5], Exit_calibrationDeltaTheta=[-2.1094217540068572E-7, 0.37625772532806073, -0.10107441100396769, -0.2751850025766889, -1.8024952768980196E-6, 2.9402326063437956E-8], Exit_calibrationA=[2.0416891277915125E-5, -0.5694828868469309, -0.5499202125525207, -9.504674691390763E-6, -3.603723657207661E-5, 0.0], Exit_calibrationD=[0.1808937726775539, -146.69166934821124, 192.91866861971778, -46.05308757405963, 0.11977780403821288, 0.11560212559305974], Exit_calibrationAlpha=[1.5714252480212174, -0.0015337665762078037, 0.0033588312559612306, 1.5687392298942362, -1.5714772428732047, 0.0], Exit_calibrationJointChecksum=[-1490546360, -1456574554, -1506622700, -1493399207, -1492840923, -1492940558], Exit_calibrationStatus=2, Exit_calibrationValidChecksum=true, Exit_baseToFeature=[0.0, 0.0, 0.0, 0.0, 0.0, 0.0], Exit_TCPOffset=[5.448621513803875E-6, -3.4480973448713925E-7, -1.4619607155264003E-5, 6.298767562616306E-5, -2.1385411919845807E-5, 2.0079116383227903E-5], currentWizardState=LANDING, Pose(key=refBaseToFeature, Position(key=posePosition, Length(key=X value=0 unit=M), Length(key=Y value=0 unit=M), Length(key=Z value=0 unit=M)), Rotation(key=poseRotation, Angle(key=RX value=0 unit=RAD), Angle(key=RY value=0 unit=RAD), Angle(key=RZ value=0 unit=RAD))), Pose(key=refPose, Position(key=posePosition, Length(key=X value=0.286405 unit=M), Length(key=Y value=-0.205786 unit=M), Length(key=Z value=0.267225 unit=M)), Rotation(key=poseRotation, Angle(key=RX value=2.177406 unit=RAD), Angle(key=RY value=-2.260348 unit=RAD), Angle(key=RZ value=0.070321 unit=RAD))), JointPositions(key=Approach_jointpositions, JointPosition(key=[1], Angle(key=pos value=-0.094237 unit=RAD)), JointPosition(key=[2], Angle(key=pos value=-1.495641 unit=RAD)), JointPosition(key=[3], Angle(key=pos value=-2.263195 unit=RAD)), JointPosition(key=[4], Angle(key=pos value=-4.063462 unit=RAD)), JointPosition(key=[5], Angle(key=pos value=-1.542982 unit=RAD)), JointPosition(key=[6], Angle(key=pos value=-3.194269 unit=RAD))), JointPositions(key=Exit_jointpositions, JointPosition(key=[1], Angle(key=pos value=-0.094265 unit=RAD)), JointPosition(key=[2], Angle(key=pos value=-1.486549 unit=RAD)), JointPosition(key=[3], Angle(key=pos value=-2.255256 unit=RAD)), JointPosition(key=[4], Angle(key=pos value=-4.080492 unit=RAD)), JointPosition(key=[5], Angle(key=pos value=-1.543016 unit=RAD)), JointPosition(key=[6], Angle(key=pos value=-3.194356 unit=RAD))))
            URCap Generated Movements (polyscope-pallet-impl, Universal Robots) state(isChildrenLocked=true)
              MoveJ speed 60 deg/s, acceleration 80 deg/s^2 (useActiveTCP=true) feature=referencePoin_6
                Waypoint Approach_5: TCP in base x=286.417 y=-205.78 z=342.031 mm, rx=2.1775 ry=-2.2603 rz=0.0702 rad; joints [-5.4, -85.696, -129.671, -232.819, -88.41, -183.02] deg; TCP offset x=0 y=0 z=0 mm, rx=0 ry=0 rz=0 rad; feature pose in base x=286.405 y=-205.786 z=267.225 mm, rx=2.1774 ry=-2.2603 rz=0.0703 rad
              MoveL speed 250 mm/s, acceleration 1200 mm/s^2 (useActiveTCP=true) feature(featureName=referencePoin_6)
                Waypoint ToolActionPoi_5: TCP in base x=286.405 y=-205.786 z=267.225 mm, rx=2.1774 ry=-2.2603 rz=0.0703 rad; joints [-5.385, -91.749, -133.659, -222.778, -88.382, -182.97] deg; TCP offset x=0 y=0 z=0 mm, rx=0 ry=0 rz=0 rad
              Folder Tool action
                URCap RG Grip (OnRobot, OnRobot A/S) dataModel(rg-target-force=40.0, rg-target-width=0.1014)
              MoveL speed 250 mm/s, acceleration 1200 mm/s^2 (useActiveTCP=true) feature(featureName=referencePoin_6)
                Waypoint Exit_6: TCP in base x=286.404 y=-205.791 z=349.6 mm, rx=2.1774 ry=-2.2604 rz=0.0704 rad; joints [-5.402, -85.171, -129.216, -233.794, -88.41, -183.024] deg; TCP offset x=0 y=0 z=0 mm, rx=0 ry=0 rz=0 rad
    Waypoint home: TCP in base x=349.211 y=-1.072 z=358.337 mm, rx=2.2343 ry=-2.1885 rz=-0.0245 rad; joints [29.524, -85.445, -128.627, -236.977, -90.829, -151.415] deg
    Halt
